// TIA Portal V17 export
// export: Created 2023-03-06T02:05:12.1760999Z, ExportSetting WithDefaults, DisplayName Totally Integrated Automation Portal, DisplayVersion V17 Update 4, DisplayName TIA Portal Openness, DisplayVersion V17 Update 4, DisplayName TIA Portal Version Control Interface, DisplayVersion V17, DisplayName STEP 7 Professional, DisplayVersion V17 Update 4, DisplayName STEP 7 Safety, DisplayVersion V17, DisplayName WinCC Professional, DisplayVersion V17 Update 4
FUNCTION "MV SKID (PE)" : Void   // FC45, LAD
TITLE = ModBus TCP for MVSKID Power Electronics
{ S7_Optimized_Access := 'TRUE' }
VERSION : 0.1
// stored: AutoNumber false, IsIECCheckEnabled false, SetENOAutomatically false, UDAEnableTagReadback false
   VAR_TEMP   // added for the SCL form of the ladder/FBD networks
      _w1 : Bool;
   END_VAR
BEGIN

REGION Network 1: Function Modbus Client
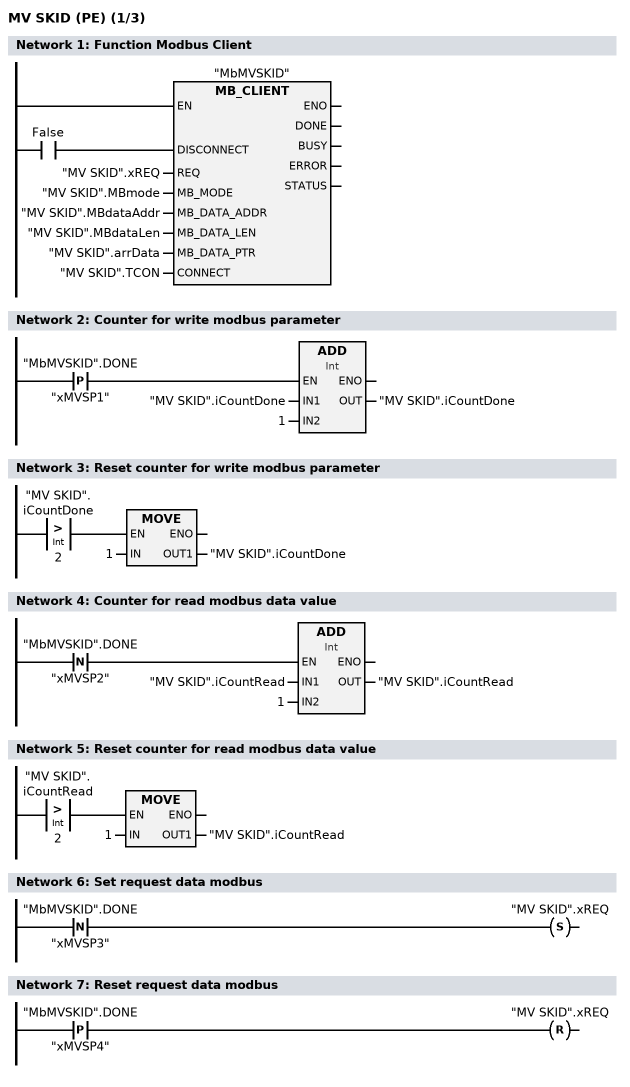
   RUNG wire#powerrail
      "MbMVSKID".MB_CLIENT(DISCONNECT := wire#w1, REQ := "MV SKID".xREQ, MB_MODE := "MV SKID".MBmode, MB_DATA_ADDR := "MV SKID".MBdataAddr, MB_DATA_LEN := "MV SKID".MBdataLen, MB_DATA_PTR := "MV SKID".arrData, CONNECT := "MV SKID".TCON, DONE =>, BUSY =>, ERROR =>, STATUS =>)
   END_RUNG
   RUNG wire#powerrail
      Contact( False )
   END_RUNG wire#w1
   // the same network as SCL:
   "MbMVSKID"(DISCONNECT := False,   // MB_CLIENT
              REQ := "MV SKID".xREQ,
              MB_MODE := "MV SKID".MBmode,
              MB_DATA_ADDR := "MV SKID".MBdataAddr,
              MB_DATA_LEN := "MV SKID".MBdataLen,
              MB_DATA_PTR := "MV SKID".arrData,
              CONNECT := "MV SKID".TCON);
END_REGION

REGION Network 2: Counter for write modbus parameter
   RUNG wire#powerrail
      P_Contact(operand := "MbMVSKID".DONE, bit := "xMVSP1")
      { S7_Templates := "SrcType := Int" } Add(in1 := "MV SKID".iCountDone, in2 := 1, out => "MV SKID".iCountDone)
   END_RUNG
   // the same network as SCL:
   #_w1 := "MbMVSKID".DONE AND NOT "xMVSP1";   // rising edge of "MbMVSKID".DONE
   "xMVSP1" := "MbMVSKID".DONE;
   IF #_w1 THEN "MV SKID".iCountDone := "MV SKID".iCountDone + 1; END_IF;
END_REGION

REGION Network 3: Reset counter for write modbus parameter
   RUNG wire#powerrail
      { S7_Templates := "SrcType := Int" } GT_Contact(in1 := "MV SKID".iCountDone, in2 := 2)
      Move(in := 1, out1 => "MV SKID".iCountDone)
   END_RUNG
   // the same network as SCL:
   IF "MV SKID".iCountDone > 2 THEN "MV SKID".iCountDone := 1; END_IF;
END_REGION

REGION Network 4: Counter for read modbus data value
   RUNG wire#powerrail
      N_Contact(operand := "MbMVSKID".DONE, bit := "xMVSP2")
      { S7_Templates := "SrcType := Int" } Add(in1 := "MV SKID".iCountRead, in2 := 1, out => "MV SKID".iCountRead)
   END_RUNG
   // the same network as SCL:
   #_w1 := NOT "MbMVSKID".DONE AND "xMVSP2";   // falling edge of "MbMVSKID".DONE
   "xMVSP2" := "MbMVSKID".DONE;
   IF #_w1 THEN "MV SKID".iCountRead := "MV SKID".iCountRead + 1; END_IF;
END_REGION

REGION Network 5: Reset counter for read modbus data value
   RUNG wire#powerrail
      { S7_Templates := "SrcType := Int" } GT_Contact(in1 := "MV SKID".iCountRead, in2 := 2)
      Move(in := 1, out1 => "MV SKID".iCountRead)
   END_RUNG
   // the same network as SCL:
   IF "MV SKID".iCountRead > 2 THEN "MV SKID".iCountRead := 1; END_IF;
END_REGION

REGION Network 6: Set request data modbus
   RUNG wire#powerrail
      N_Contact(operand := "MbMVSKID".DONE, bit := "xMVSP3")
      S_Coil( "MV SKID".xREQ )
   END_RUNG
   // the same network as SCL:
   #_w1 := NOT "MbMVSKID".DONE AND "xMVSP3";   // falling edge of "MbMVSKID".DONE
   "xMVSP3" := "MbMVSKID".DONE;
   IF #_w1 THEN "MV SKID".xREQ := TRUE; END_IF;
END_REGION

REGION Network 7: Reset request data modbus
   RUNG wire#powerrail
      P_Contact(operand := "MbMVSKID".DONE, bit := "xMVSP4")
      R_Coil( "MV SKID".xREQ )
   END_RUNG
   // the same network as SCL:
   #_w1 := "MbMVSKID".DONE AND NOT "xMVSP4";   // rising edge of "MbMVSKID".DONE
   "xMVSP4" := "MbMVSKID".DONE;
   IF #_w1 THEN "MV SKID".xREQ := FALSE; END_IF;
END_REGION

REGION Network 8: Write R_MVSKID parameter
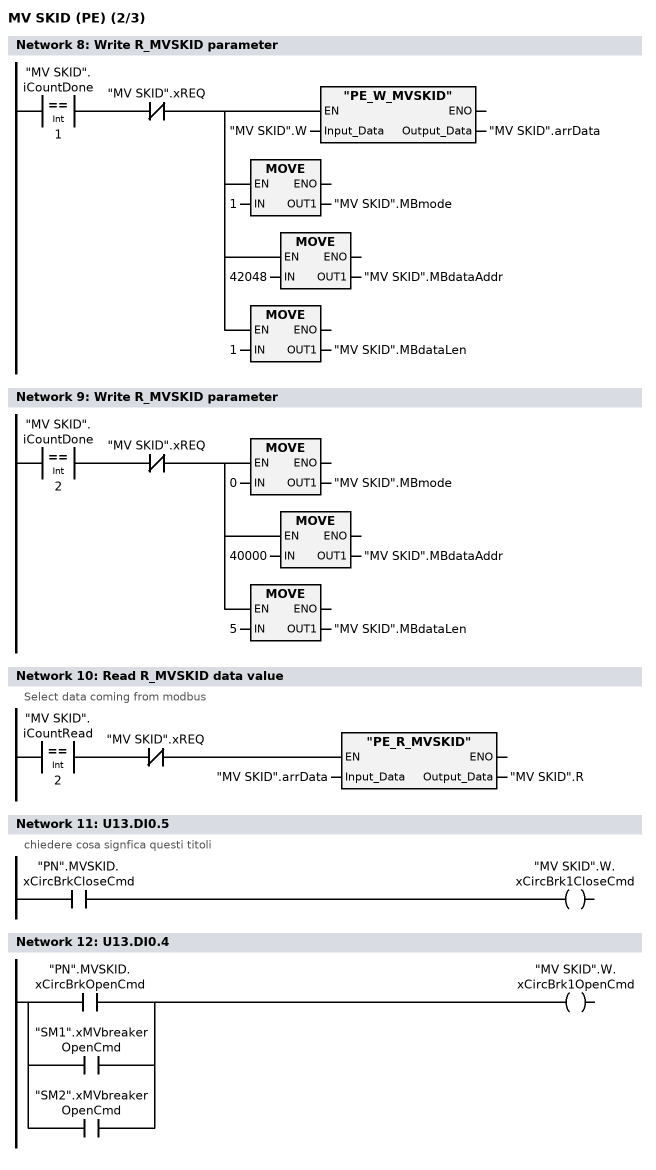
   RUNG wire#powerrail
      { S7_Templates := "SrcType := Int" } EQ_Contact(in1 := "MV SKID".iCountDone, in2 := 1)
      I_Contact( "MV SKID".xREQ )
      wire#w1
      "PE_W_MVSKID"(Input_Data := "MV SKID".W, Output_Data => "MV SKID".arrData)
   END_RUNG
   RUNG wire#w1
      Move(in := 1, out1 => "MV SKID".MBmode)
   END_RUNG
   RUNG wire#w1
      Move(in := 42048, out1 => "MV SKID".MBdataAddr)
   END_RUNG
   RUNG wire#w1
      Move(in := 1, out1 => "MV SKID".MBdataLen)
   END_RUNG
   // the same network as SCL:
   #_w1 := ("MV SKID".iCountDone = 1) AND NOT "MV SKID".xREQ;
   IF #_w1 THEN
       "PE_W_MVSKID"(Input_Data := "MV SKID".W, Output_Data => "MV SKID".arrData);
       "MV SKID".MBmode := 1;
       "MV SKID".MBdataAddr := 42048;
       "MV SKID".MBdataLen := 1;
   END_IF;
END_REGION

REGION Network 9: Write R_MVSKID parameter
   RUNG wire#powerrail
      { S7_Templates := "SrcType := Int" } EQ_Contact(in1 := "MV SKID".iCountDone, in2 := 2)
      I_Contact( "MV SKID".xREQ )
      wire#w1
      Move(in := 0, out1 => "MV SKID".MBmode)
   END_RUNG
   RUNG wire#w1
      Move(in := 40000, out1 => "MV SKID".MBdataAddr)
   END_RUNG
   RUNG wire#w1
      Move(in := 5, out1 => "MV SKID".MBdataLen)
   END_RUNG
   // the same network as SCL:
   IF ("MV SKID".iCountDone = 2) AND NOT "MV SKID".xREQ THEN
       "MV SKID".MBmode := 0;
       "MV SKID".MBdataAddr := 40000;
       "MV SKID".MBdataLen := 5;
   END_IF;
END_REGION

REGION Network 10: Read R_MVSKID data value
   // Select data coming from modbus
   RUNG wire#powerrail
      { S7_Templates := "SrcType := Int" } EQ_Contact(in1 := "MV SKID".iCountRead, in2 := 2)
      I_Contact( "MV SKID".xREQ )
      "PE_R_MVSKID"(Input_Data := "MV SKID".arrData, Output_Data => "MV SKID".R)
   END_RUNG
   // the same network as SCL:
   IF ("MV SKID".iCountRead = 2) AND NOT "MV SKID".xREQ THEN
       "PE_R_MVSKID"(Input_Data := "MV SKID".arrData, Output_Data => "MV SKID".R);
   END_IF;
END_REGION

REGION Network 11: U13.DI0.5
   // chiedere cosa signfica questi titoli
   RUNG wire#powerrail
      Contact( "PN".MVSKID.xCircBrkCloseCmd )
      Coil( "MV SKID".W.xCircBrk1CloseCmd )
   END_RUNG
   // the same network as SCL:
   "MV SKID".W.xCircBrk1CloseCmd := "PN".MVSKID.xCircBrkCloseCmd;
END_REGION

REGION Network 12: U13.DI0.4
   RUNG wire#powerrail
      Contact( "PN".MVSKID.xCircBrkOpenCmd )
      wire#w1
      Coil( "MV SKID".W.xCircBrk1OpenCmd )
   END_RUNG
   RUNG wire#powerrail
      Contact( "SM1".xMVbreakerOpenCmd )
   END_RUNG wire#w1
   RUNG wire#powerrail
      Contact( "SM2".xMVbreakerOpenCmd )
   END_RUNG wire#w1
   // the same network as SCL:
   "MV SKID".W.xCircBrk1OpenCmd := "PN".MVSKID.xCircBrkOpenCmd OR "SM1".xMVbreakerOpenCmd OR "SM2".xMVbreakerOpenCmd;
END_REGION

REGION Network 13: MV SKID Fault
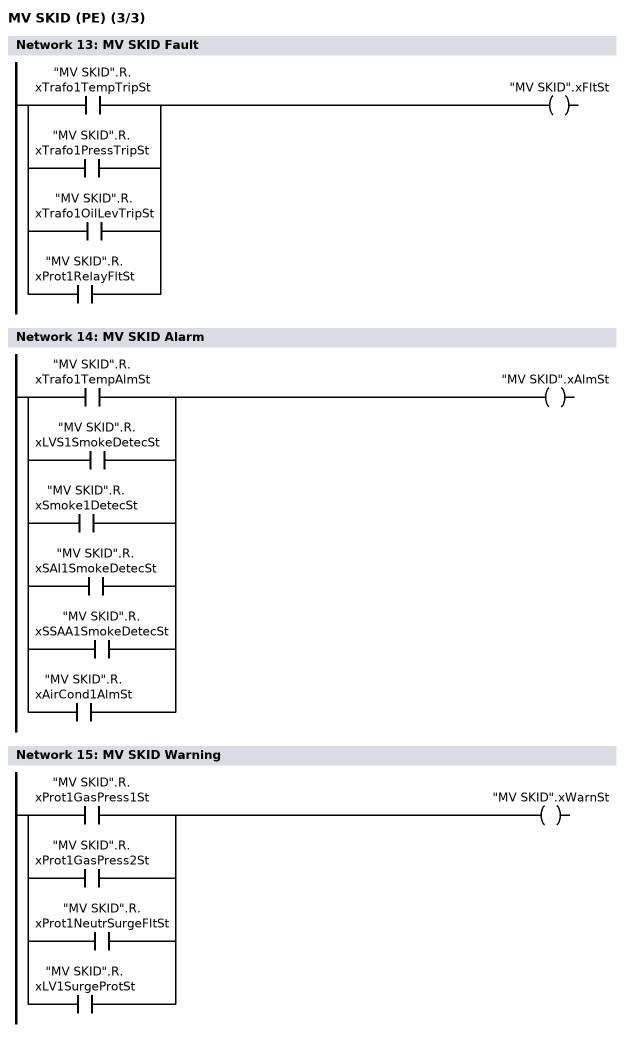
   RUNG wire#powerrail
      Contact( "MV SKID".R.xTrafo1TempTripSt )
      wire#w1
      Coil( "MV SKID".xFltSt )
   END_RUNG
   RUNG wire#powerrail
      Contact( "MV SKID".R.xTrafo1PressTripSt )
   END_RUNG wire#w1
   RUNG wire#powerrail
      Contact( "MV SKID".R.xTrafo1OilLevTripSt )
   END_RUNG wire#w1
   RUNG wire#powerrail
      Contact( "MV SKID".R.xProt1RelayFltSt )
   END_RUNG wire#w1
   // the same network as SCL:
   "MV SKID".xFltSt := "MV SKID".R.xTrafo1TempTripSt OR "MV SKID".R.xTrafo1PressTripSt OR "MV SKID".R.xTrafo1OilLevTripSt OR "MV SKID".R.xProt1RelayFltSt;
END_REGION

REGION Network 14: MV SKID Alarm
   RUNG wire#powerrail
      Contact( "MV SKID".R.xTrafo1TempAlmSt )
      wire#w1
      Coil( "MV SKID".xAlmSt )
   END_RUNG
   RUNG wire#powerrail
      Contact( "MV SKID".R.xLVS1SmokeDetecSt )
   END_RUNG wire#w1
   RUNG wire#powerrail
      Contact( "MV SKID".R.xSmoke1DetecSt )
   END_RUNG wire#w1
   RUNG wire#powerrail
      Contact( "MV SKID".R.xSAI1SmokeDetecSt )
   END_RUNG wire#w1
   RUNG wire#powerrail
      Contact( "MV SKID".R.xSSAA1SmokeDetecSt )
   END_RUNG wire#w1
   RUNG wire#powerrail
      Contact( "MV SKID".R.xAirCond1AlmSt )
   END_RUNG wire#w1
   // the same network as SCL:
   "MV SKID".xAlmSt := "MV SKID".R.xTrafo1TempAlmSt OR "MV SKID".R.xLVS1SmokeDetecSt OR "MV SKID".R.xSmoke1DetecSt OR "MV SKID".R.xSAI1SmokeDetecSt OR "MV SKID".R.xSSAA1SmokeDetecSt OR "MV SKID".R.xAirCond1AlmSt;
END_REGION

REGION Network 15: MV SKID Warning
   RUNG wire#powerrail
      Contact( "MV SKID".R.xProt1GasPress1St )
      wire#w1
      Coil( "MV SKID".xWarnSt )
   END_RUNG
   RUNG wire#powerrail
      Contact( "MV SKID".R.xProt1GasPress2St )
   END_RUNG wire#w1
   RUNG wire#powerrail
      Contact( "MV SKID".R.xProt1NeutrSurgeFltSt )
   END_RUNG wire#w1
   RUNG wire#powerrail
      Contact( "MV SKID".R.xLV1SurgeProtSt )
   END_RUNG wire#w1
   // the same network as SCL:
   "MV SKID".xWarnSt := "MV SKID".R.xProt1GasPress1St OR "MV SKID".R.xProt1GasPress2St OR "MV SKID".R.xProt1NeutrSurgeFltSt OR "MV SKID".R.xLV1SurgeProtSt;
END_REGION

REGION Network 16 (SCL): MV SKID Line Disconnector & Breaker Status
   "MV SKID".wLine1DiscSt.%X0 := "MV SKID".R.xLine1DiscOpenSt;
   "MV SKID".wLine1DiscSt.%X1 := "MV SKID".R.xLine1DiscCloseSt;
   "MV SKID".wLine1DiscSt.%X2 := "MV SKID".R.xLine1GndCloseSt;

   "MV SKID".wLine2DiscSt.%X0 := "MV SKID".R.xLine2DiscOpenSt;
   "MV SKID".wLine2DiscSt.%X1 := "MV SKID".R.xLine2DiscCloseSt;
   "MV SKID".wLine2DiscSt.%X2 := "MV SKID".R.xLine2GndCloseSt;

   "MV SKID".wProt1DiscSt.%X0 := "MV SKID".R.xProt1DiscOpenSt;
   "MV SKID".wProt1DiscSt.%X1 := "MV SKID".R.xProt1DiscCloseSt;
   "MV SKID".wProt1DiscSt.%X2 := "MV SKID".R.xProt1GndCloseSt;

   "MV SKID".wProt1CircBrkSt.%X0 := "MV SKID".R.xProt1CircBrkOpenSt;
   "MV SKID".wProt1CircBrkSt.%X1 := "MV SKID".R.xProt1CircBrkCloseSt;
END_REGION
END_FUNCTION
